PROGRAM MAIN
VAR
END_VAR


prgAlarmHnd();

END_PROGRAM

(* stored: Version 1.1.0.1
   POU MAIN: Id {049bc518-a29e-4463-8c79-418e3c1a10e6}, SpecialFunc None *)
